TYPE "UDT_MOTOR"
VERSION : 0.1
   STRUCT
      RUN_FEEDBACK : BOOL;
      SPEED : REAL;
   END_STRUCT;

END_TYPE
